
// ===== library: MasterCopy "FifoQueueHandler" =====

FUNCTION_BLOCK "FifoQueueHandler"   // FB1, SCL
{ S7_Optimized_Access := 'TRUE' }
VERSION : 0.1
   VAR_INPUT
      DataIn : "FifoStruct";
   END_VAR
   VAR_OUTPUT
      DataQ : Array[0..19] of Bool;
   END_VAR
   VAR
      ChannelData : Array[0..19] of "FifoStruct";
      InQueue : Array[0..19] of Bool;
      QueueSize : Int;
      FifoIndex : Int;
      ScanIndex : Int;
      QueueLength : Int;
      MaxActiveRequests : Int;
      i : Int;
      j : Int;
   END_VAR
BEGIN
   (*
    // -----------------------------------------------------------------------------
    // LICENSE:
    //  Released under the MIT License
    //  Copyright (c) 2025 Jesús Alguacil
    //  Full license text available at:
    //  https://github.com/JessAlguacil/FifoQueueHandler/blob/master/LICENSE.md
    // -----------------------------------------------------------------------------
    // Function      : FifoQueueHandler
    // Description   : Generic FIFO queue handler that activates a limited number of simultaneous requests.
                       Processes distributed input channels using a circular index,
                       queues new requests, activates a limited number at a time,
                       and removes those that are no longer active.

    // Compatibility : IEC 61131-3 (Structured Text)
    // Author        : Jesús Alguacil
    // Date          : 28/06/2025
    // Version       : 1.2
    // -----------------------------------------------------------------------------

    // GENERAL FUNCTIONALITY:
    // - Evaluates one input request per scan using a circular scan index.
    // - Adds new requests to a FIFO queue if not already queued.
    // - Activates up to a configurable number of requests simultaneously.
    // - Removes entries from the queue if the corresponding input becomes inactive.
    // - Ensures that each input can only exist once in the queue (no duplication).

    // PERFORMANCE OPTIMIZATION:
    // - Evaluates only 1 input per scan cycle → significantly reduces CPU usage.
    // - Especially suitable for large-scale input handling (e.g., 20+ channels).
    // - FIFO logic is distributed across cycles for smoother real-time performance.

    // MAIN LOGIC:
    // - STEP 1: Process input at current ScanIndex and add to queue if eligible.
    // - STEP 2: Activate the first N requests in the FIFO queue.
    // - STEP 3: Remove requests from the queue if the input becomes inactive.

    // INPUT STRUCTURE:
    // - DataIn.QueueLength           → Maximum number of entries allowed in the queue.
    // - DataIn.MaxActiveRequests     → Maximum simultaneous active requests (e.g., 3).
    // - DataIn.Input[0..N-1]         → BOOL array of input request signals.

    // OUTPUTS:
    // - DataQ[0..N-1]                → BOOL array of output activation signals.
    // - QueueSize                    → Current number of items in the queue.
    // - ChannelData[].Active         → TRUE if the channel is currently active.

    // INTERNALS:
    // - ChannelData[].Request        → Captures input request state.
    // - ChannelData[].Queue          → Stores index of the input in FIFO order.
    // - InQueue[0..N-1]              → Flags to prevent duplicate queuing.
    // - ScanIndex                    → Circular index that defines which input is evaluated this scan.
    // - FifoIndex                    → Index used for accessing items in queue.

    // NOTES:
    // - Designed for efficient real-time control in industrial applications.
    // - Generic structure supports any type of request source: motors, valves, stations, etc.
    // - Can be expanded to support priorities, timeouts, or dynamic configuration via HMI.
    // -----------------------------------------------------------------------------
   *)


   (*-------------------------------------------------------------------------------
   // STEP 1: PROCESS NEW REQUESTS AND ADD TO THE QUEUE IF NOT ALREADY QUEUED
   ---------------------------------------------------------------------------------*)

   // Read input parameters
   #QueueLength := #DataIn.QueueLength;
   #MaxActiveRequests := #DataIn.MaxActiveRequests;

   // Update request and input status
   #ChannelData[#ScanIndex].Request := #DataIn.Input[#ScanIndex];
   #DataQ[#ScanIndex] := #ChannelData[#ScanIndex].Active;

   // Counter that scans the FIFO index
   #ScanIndex := (#ScanIndex + 1) MOD #QueueLength;

   IF #ChannelData[#ScanIndex].Request AND NOT #InQueue[#ScanIndex] AND #QueueSize < #QueueLength THEN
       #QueueSize := #QueueSize + 1;
       #ChannelData[#QueueSize].Queue := #ScanIndex;
       #InQueue[#ScanIndex] := TRUE;
   END_IF;

   // Reset outputs
   #ChannelData[#ScanIndex].Active := FALSE;


   (*-------------------------------------------------------------------------------
   // STEP 2: ACTIVATE ONLY THE FIRST NUMBERS MOTORS IN THE QUEUE
   ---------------------------------------------------------------------------------*)

   FOR #i := 0 TO MIN(IN1:=#MaxActiveRequests-1, IN2:= #QueueSize) DO
       #FifoIndex := #ChannelData[#i].Queue;
       #ChannelData[#FifoIndex].Active := TRUE;
   END_FOR;

   (*-------------------------------------------------------------------------------
   // STEP 3: REMOVE FROM QUEUE THE MOTORS THAT ARE NO LONGER REQUESTING
   ---------------------------------------------------------------------------------*)

   #i := 0;
   WHILE #i <= #QueueSize DO
       #FifoIndex := #ChannelData[#i].Queue;
       IF NOT #ChannelData[#FifoIndex].Request THEN
           // Shift elements left
           FOR #j := #i TO #QueueSize - 1 DO
               #ChannelData[#j].Queue := #ChannelData[#j + 1].Queue;
           END_FOR;

           #QueueSize := #QueueSize - 1;
           #InQueue[#FifoIndex] := FALSE;

           // Don't increment i, since new item is now in the same position
       ELSE
           #i := #i + 1;
       END_IF;
   END_WHILE;

   // END BLOCK
END_FUNCTION_BLOCK

// ===== library: MasterCopy "FifoStruct" =====

TYPE "FifoStruct"
   STRUCT
      Request : Bool;
      Active : Bool;
      Queue : Int;
      QueueLength : Int;
      MaxActiveRequests : Int;
      Input : Array[0..19] of Bool;
   END_STRUCT;
END_TYPE